TYPE ST_Wash :
STRUCT
	nWaterLevel : INT ;
	eWashStrategy : E_Strategy;
	
END_STRUCT
END_TYPE

(* stored: Version 1.1.0.1, ProductVersion 3.1.4024.16
   DUT ST_Wash: Id {8ae3c9b4-99f1-4974-9113-2b578a6d7aa1} *)
